# EPICS autosave request: ipApp/Db/AE_ILS_settings.req
# FILE...AE_ILS_settings.req

$(P)$(R)VoltMeas.SCAN
$(P)$(R)VoltMeas.DESC
$(P)$(R)Volt
$(P)$(R)VoltTweakVal
$(P)$(R)VoltLimit
$(P)$(R)Current
$(P)$(R)CurrentTweakVal
$(P)$(R)CurrentLimit
$(P)$(R)Power
$(P)$(R)PowerTweakVal
$(P)$(R)PowerLimit
